{attribute 'qualified_only'}
VAR_GLOBAL
    testAxis : AXIS_REF;
END_VAR

(* stored: Version 1.1.0.1
   GVL NcAxis_GVL: Id {c2946879-f813-4e4a-acb0-1c588477f389} *)
